RoboDK station: Celda robotizada DRILLING.rdk

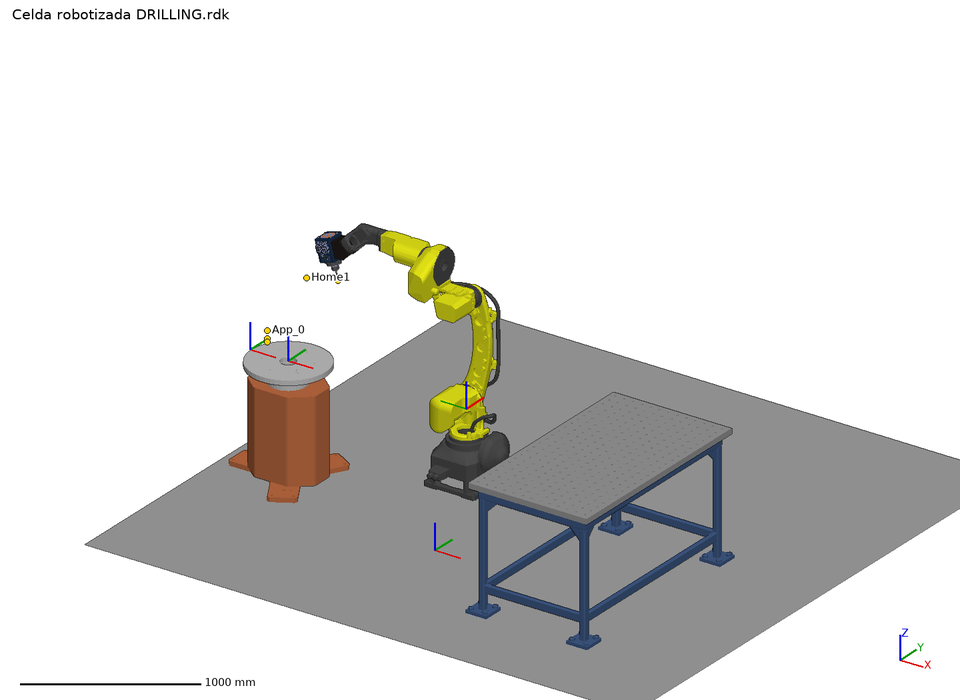
[picture v0: the station drawn from its stored meshes, robots at their saved joint values, targets as dots, program paths as lines]
Station Celda robotizada DRILLING (saved by RoboDK 5.9.3). Poses are relative to the parent item; angles as X-Y-Z fixed-axis rotations.
  - frame Fanuc M-10iD/12 Base at (0, 300, 750) mm, rotated rx 0 ry 0 rz 90 deg
    - robot Fanuc M-10iD/12: 6 axes, payload 12 kg, reach 1441 mm, repeatability 0.02 mm, weight 145 kg
        modified DH rows (alpha deg, a mm, theta deg, d mm): 0, 0, 0, 450; -90, 75, -90, 0; 0, 640, 0, 0; -90, 195, 0, 700; 90, 0, 0, 0; -90, 0, 0, 75
        base shift (0, 0, -450) mm
        joint limits [-170, -90, -95, -190, -190, -450] to [170, 160, 180, 190, 190, 450]; home [2.41, -13.166, -36.386, 2.747, 36.42, 179.892]; saved at [90.871, -3.548, 0.989, 0.856, -45.995, 178.79]
      - tool Custom Spindle, TCP at (118.9, 0, 221.26) mm, rotated rx 60 ry 0 rz 90 deg, size 260.9 x 152 x 222 mm, geometry from KUKA KP1-V 500 Base
    - target Home1 (joint target) at (-11.12, 1067.72, 509.95) mm, rotated rx 180 ry 0 rz -90 deg; joints [90.871, -3.548, 0.989, 0.856, -45.995, 178.79] of Fanuc M-10iD/12
  - frame KUKA KP1-V 500 Base at (-1200, 300, 710) mm
    - robot KUKA KP1-V 500: 1 axes, payload 500 kg
        modified DH rows (alpha deg, a mm, theta deg, d mm): 0, 0, 0, 0
        joint limits [-720] to [720]; home [0]; saved at [0]
      - frame CAD_Frame at (-172.52, -117.59, 66.56) mm
        - target Home (joint target) at (515.26, 106.46, 525.71) mm, rotated rx -165 ry 0 rz -90 deg; joints [90.871, -3.548, 0.989, 0.856, -45.995, 178.79] of Fanuc M-10iD/12
        - target App_0 (Cartesian target) at (25, 125, 75) mm, rotated rx -180 ry 0 rz 180 deg; joints [9.435, -11.391, -0.256, -9.269, -133.978, 346.833] of Fanuc M-10iD/12
        - target Pos_0 (Cartesian target) at (25, 125, 25) mm, rotated rx -180 ry 0 rz 180 deg; joints [9.435, -11.391, -0.256, -9.269, -133.978, 346.833] of Fanuc M-10iD/12
        - target Deep_0 (Cartesian target) at (25, 125, 5) mm, rotated rx -180 ry 0 rz 180 deg; joints [9.435, -11.391, -0.256, -9.269, -133.978, 346.833] of Fanuc M-10iD/12
    - target P1 (Cartesian target) at (172.52, 117.59, -66.56) mm; joints [0] of KUKA KP1-V 500
  - frame World at (0, 0, 0) mm
    - object Table 1400x800x800mm at (1000, -200, 800) mm, rotated rx 0 ry 0 rz 90 deg, size 1420 x 820 x 800 mm, geometry from Table-1400x800x800mm.sld
    - object Floor at (570, 450, 0) mm, size 3000 x 3000 x 0 mm, geometry from Floor.sld
      - object Floor at (-700, 0, 0) mm, size 3000 x 3000 x 0 mm, geometry from Floor.sld
      - object Floor at (0, 650, 0) mm, size 3000 x 3000 x 0 mm, geometry from Floor.sld
        - object Floor at (-700, 0, 0) mm, size 3000 x 3000 x 0 mm, geometry from Floor.sld
    - object RoboticCell_v1 at (-390, -940, 0) mm, geometry from RoboticCell_v1.step
      - item type 7 RoboticCell_v1-21
      - item type 7 RoboticCell_v1-22
      - item type 7 RoboticCell_v1-23
      - item type 7 RoboticCell_v1-24
      - item type 7 RoboticCell_v1-28
      - item type 7 RoboticCell_v1-29
      - item type 7 RoboticCell_v1-30
      - item type 7 RoboticCell_v1-31
      - item type 7 RoboticCell_v1-32
      - item type 7 RoboticCell_v1-33
      - item type 7 RoboticCell_v1-34
      - item type 7 RoboticCell_v1-35
      - item type 7 RoboticCell_v1-36
      - item type 7 RoboticCell_v1-38
      - item type 7 RoboticCell_v1-46
      - item type 7 RoboticCell_v1-47
      - item type 7 RoboticCell_v1-48
      - item type 7 RoboticCell_v1-27
      - item type 7 RoboticCell_v1-26
      - item type 7 RoboticCell_v1-25
